// TwinCAT 3 PLC project CORE
// Title: Core
// Company: Ziga
// Author: Ziga Javornik
// ProjectVersion: 0.0.0.1
// Description: A collection of core objects for work with further libraries implementations.
// ProgramVersion: 3.1.4024.0
// libraries:
//   Tc2_Standard, * (Beckhoff Automation GmbH)
//   Tc2_System, * (Beckhoff Automation GmbH)
//   Tc2_Utilities, * (Beckhoff Automation GmbH)
//   Tc3_Module, * (Beckhoff Automation GmbH)
//   TcUnit, * (www.tcunit.org)
// project tree:
//   SOURCE/Ams/Helpers/ AmsHelper.TcPOU (not stored)
//   SOURCE/Ams/ITFs/ I_RequiresAmsAddress.TcIO (not stored)
//   SOURCE/Array/ ArrayHelper.TcPOU (not stored)
//   SOURCE/File/DUTs/ ST_FileProperties.TcDUT
//   SOURCE/File/Helpers/ FileHelper.TcPOU (not stored)
//   SOURCE/File/ITFs/ I_FileProperties.TcIO (not stored)
//   SOURCE/Logger/DUTs/ ST_LogLevelHeaders.TcDUT (not stored)
//   SOURCE/Logger/ITFs/ I_Logger.TcIO (not stored), I_LoggerEx.TcIO (not stored)
//   SOURCE/String/Helpers/ StringHelper.TcPOU (not stored)
//   SOURCE/String/ITFs/ I_StringBuilder.TcIO (not stored)
//   SOURCE/String/POUs/ FB_StringBuilderBase.TcPOU (not stored), StringConstants.TcPOU (not stored)
//   SOURCE/Time/DUTs/ E_TimeFormat.TcDUT, ST_CurrentSystemTimeInfo.TcDUT (not stored)
//   SOURCE/Time/Helpers/ TimeHelper.TcPOU (not stored)
//   SOURCE/Time/POUs/ FB_LocalSystemTimeProvider.TcPOU (not stored)
//   / TestsTask.TcTTO (not stored)
//   TESTS/ PRG_TESTS.TcPOU (not stored)
//   TESTS/Test suites/ FB_AmsHelper_Tests.TcPOU
// (motion and I/O tree: see PLC project io)
// real-time tasks:
//   TASK TestsTask: cycle T#10ms, priority 20, ADS port 350

// ---- SOURCE/File/DUTs/ST_FileProperties.TcDUT
TYPE ST_FileProperties :
STRUCT
	FileLocation 	: Tc2_System.T_MaxString;
	FileName		: Tc2_System.T_MaxString;
END_STRUCT
END_TYPE

// ---- SOURCE/Time/DUTs/E_TimeFormat.TcDUT
{attribute 'qualified_only'}
{attribute 'strict'}
TYPE E_TimeFormat :
(
	HHMMSS,
	DDMMYY,
	YYMMDD,
	MMDDYY,
	DDMMYY_HHMMSS,
	YYMMDD_HHMMSS,
	MMDDYY_HHMMSS
);
END_TYPE

// ---- TESTS/Test suites/FB_AmsHelper_Tests.TcPOU
// Subject under test
FUNCTION_BLOCK FB_AmsHelper_Tests EXTENDS FB_TestSuite

// Create instance variables that will be accesible for all tests
VAR
END_VAR

// Call your test methods here
THIS^.Test_EmptyNetId_ExpectEmptyString();

METHOD PRIVATE Test_EmptyNetId_ExpectEmptyString

(* Instanced variables are VERY useful for writing tests since tests are run in paralel (by default).
By instantiating local variables that are not placed on the same stack as method (values are retained between calls)
you make sure that the SUT is not changed by some other test. *)
VAR_INST
	
END_VAR

// Place temporary variables here
VAR
	emptyNetId	: Tc2_System.T_AmsNetIdArr;
END_VAR
// The name of the test, is the same as method name!
TcUnit.TEST('Test_EmptyNetId_ExpectEmptyString');

// Do your assertions here...
AssertEquals_STRING(
	Expected := '',
	Actual := AmsHelper.NetIdToString(emptyNetId),
	Message := 'An empty netId should return an empty string!');

TcUnit.TEST_FINISHED();
END_METHOD

END_FUNCTION_BLOCK
